PROGRAM Log_Csv
VAR
	trig1 : BOOL := FALSE;
	// Trang thai cho su kien
	eEventType : E_EventType := E_EventType.Alarm;
	eEventSeverity : TcEventSeverity := TcEventSeverity.Error;
	nEventIdentity : UDINT := 32;
	sEventText : STRING(255) := 'Status';
	nEventID : UDINT;
	
	CsvPersistentEventStorage : FB_CsvPersistentEventStorage;
	EventLogger : EventLogger(CsvPersistentEventStorage);
END_VAR


IF trig1 THEN
    // Gọi method GetEventTextByID từ CsvPersistentEventStorage để lấy text dựa trên nEventID
    sEventText := CsvPersistentEventStorage.GetEventTextByID(nEventID);
    // Ghi log sự kiện với thông tin đã cập nhật
    EventLogger.AddEvent(eEventType, eEventSeverity, nEventIdentity, sEventText);
    trig1 := FALSE;
END_IF;
CsvPersistentEventStorage();

END_PROGRAM

(* stored: Version 1.1.0.1, ProductVersion 3.1.4024.12
   POU Log_Csv: Id {0ee1b1a8-85cb-4141-a608-07f7a6b247ce}, SpecialFunc None *)
